(* CODESYS project Tc3_XtsInterface.library
   TcLibraryId: Beckhoff Automation GmbH|Tc3_XtsInterface|0.2.15.0
   Company: Beckhoff Automation GmbH
   Title: Tc3_XtsInterface
   Version: 0.2.15.0

Project tree, tasks and I/O mapping:
  POUs/
    Environment/
      ProcessingUnit/
        Mover/
          function block FB_XtsXlMover [ST]: FB_init, FB_exit, Init, GetParameter, SetParameter, GetObjectId, Environment, ProcessingUnit, GetActiveTrackObjectId, SetActiveTrackObjectId, GetConfiguredDetectionTrackObjectId, SetConfiguredDetectionTrackObjectId, GetStartupTrackPosition, SetStartupTrackPosition, TriggerLeave, TriggerArrive, GetSimulatedStartUpPart, SetSimulatedStartUpPart, GetSimulatedStartUpPosition, SetSimulatedStartUpPosition, GetIsVirtualFeedbackEnabled, SetIsVirtualFeedbackEnabled, GetIsDetectionOnStartupEnabled, GetIsActive, GetPositionInfo_partPosition, GetPositionInfo_trackPosition, GetPositionInfo_partObjectId, GetPositionInfo_trackObjectId, GetBtn, GetCurrentModuleCount, GetAxisId, GetAxisObjectId, GetDistanceDriven, GetDistanceDrivenInKm, GetHasDriveError, GetMoverControllerError, GetDriveStatus, GetDriveControlValue, GetMoverController, SetMoverController, GetVersion_Major, GetVersion_Minor, GetVersion_Build, GetVersion_Revision
        Part/
          Module/
            function block FB_XtsXlModule [ST]: FB_init, FB_exit, Init, GetParameter, SetParameter, GetObjectId, Environment, Part, GetIsDcLinkVoltageReady, GetVersion_Major, GetVersion_Minor, GetVersion_Build, GetVersion_Revision
          function block FB_XtsXlPart [ST]: FB_init, FB_exit, Init, GetParameter, SetParameter, GetObjectId, Environment, ModuleCount, Module, ModuleWithOid, ProcessingUnit, GetMcTrackOid, GetLength, TriggerReset, GetIsDcLinkVoltageReady, GetDriveState, GetGlobalNumber, GetVersion_Major, GetVersion_Minor, GetVersion_Build, GetVersion_Revision
        Track/
          function block FB_XtsTrack [ST]: FB_init, FB_exit, Init, GetParameter, SetParameter, GetObjectId, Environment, PartConfigCount, GetPartConfigOidAt, ProcessingUnit, GetIsClosed, GetPolarity, GetOffset, GetIsIncludedInDetection, GetDetectionPriority, GetLength, GetVersion_Major, GetVersion_Minor, GetVersion_Build, GetVersion_Revision
        function block FB_XtsProcessingUnit [ST]: FB_init, FB_exit, Init, GetParameter, SetParameter, GetObjectId, Environment, XlMoverCount, XlMover, XlMoverWithOid, XlPartCount, XlPart, XlPartWithOid, TrackCount, Track, TrackWithOid, GetActiveMoverCount, GetDriveState, GetIsDcLinkVoltageReady, GetVersion_Major, GetVersion_Minor, GetVersion_Build, GetVersion_Revision
      function block FB_XtsEnvironment [ST]: FB_init, FB_exit, Init, ProcessingUnitCount, ProcessingUnit, ProcessingUnitWithOid
  Version/
    global variables Global_Version
*)

// Version/Global_Version
{attribute 'TcGenerated'}
// This function has been automatically generated from the project information.
VAR_GLOBAL CONSTANT
	{attribute 'const_non_replaced'}
	{attribute 'linkalways'}
	stLibVersion_Tc3_XtsInterface : ST_LibVersion := (iMajor := 0, iMinor := 2, iBuild := 15, iRevision := 0, nFlags := 0, sVersion := '0.2.15.0');
	{attribute 'const_non_replaced'}
	{attribute 'linkalways'}
	sLibraryId_Tc3_XtsInterface : String := 'Beckhoff Automation GmbH|Tc3_XtsInterface|0.2.15.0';
END_VAR

// POUs/Environment/FB_XtsEnvironment

{attribute 'c++_compatible'}
{attribute 'external_name' := 'FB_XtsEnvironment_GUID_43DC2321_88A6_68C5_F281_B52FDA472D50'}
{attribute 'TcIecLibraryType'}
FUNCTION_BLOCK FB_XtsEnvironment
VAR
	 {attribute 'hide'}
	_reserved1 : ARRAY [1..12] OF UINT_8_16;
END_VAR

{attribute 'TcTypeSystem'}

(* Internal method *)
{attribute 'hide'}
METHOD FB_init : BOOL
VAR_INPUT
	(* If TRUE, the retain variables are initialized (warm start / cold start) *)
	bInitRetains : BOOL;
	(* If TRUE, the instance afterwards gets moved into the copy code (online change) *)
	bInCopyCode : BOOL;
END_VAR
END_METHOD

{attribute 'TcTypeSystem'}

(* Internal method *)
{attribute 'hide'}
METHOD FB_exit : BOOL
VAR_INPUT
	(* If TRUE, the exit method is called for exiting an instance that is copied afterwards (online change). *)
	bInCopyCode : BOOL;
END_VAR
END_METHOD

{attribute 'TcTypeSystem'}

(* Initialize the XTS environment. *)
METHOD Init
VAR_INPUT
	(* Feedback for the command. Use 0 if no feedback wanted. *)
	{attribute 'GUID' := '5F1A75BA-B0CF-46E4-B9FF-8350B6E0F16A'}
	{attribute 'Namespace' := 'Tc3_XtsInterface'}
	CommandFeedback : REFERENCE TO XtsCommandFeedback;
END_VAR
END_METHOD

{attribute 'TcTypeSystem'}

(* Returns the count of the Processing Units in the Environment. *)
METHOD ProcessingUnitCount : UINT
END_METHOD

{attribute 'TcTypeSystem'}

(* Returns the I_XtsProcessingUnit at the specified index [1, ..., size] in the Environment. *)
METHOD ProcessingUnit : I_XtsProcessingUnit1
VAR_INPUT
	(* Index of the ProcessingUnit in the Environment [1, ..., size]. *)
	Index : UINT;
	(* Feedback for the command. Use 0 if no feedback wanted. *)
	{attribute 'GUID' := '5F1A75BA-B0CF-46E4-B9FF-8350B6E0F16A'}
	{attribute 'Namespace' := 'Tc3_XtsInterface'}
	CommandFeedback : REFERENCE TO XtsCommandFeedback;
END_VAR
END_METHOD

{attribute 'TcTypeSystem'}

(* Returns the I_XtsProcessingUnit with the specified Object ID. *)
METHOD ProcessingUnitWithOid : I_XtsProcessingUnit1
VAR_INPUT
	(* Index of the ProcessingUnit in the Environment [1, ..., size]. *)
	{attribute 'GUID' := '18071995-0000-0000-0000-00000000000F'}
	ObjectId : GLOBAL.OTCID;
	(* Feedback for the command. Use 0 if no feedback wanted. *)
	{attribute 'GUID' := '5F1A75BA-B0CF-46E4-B9FF-8350B6E0F16A'}
	{attribute 'Namespace' := 'Tc3_XtsInterface'}
	CommandFeedback : REFERENCE TO XtsCommandFeedback;
END_VAR
END_METHOD

END_FUNCTION_BLOCK

// POUs/Environment/ProcessingUnit/FB_XtsProcessingUnit

{attribute 'c++_compatible'}
{attribute 'external_name' := 'FB_XtsProcessingUnit_GUID_11AFE61A_C1C5_6F5D_D8AE_C0074E97D741'}
{attribute 'TcIecLibraryType'}
FUNCTION_BLOCK FB_XtsProcessingUnit
VAR
	 {attribute 'hide'}
	_reserved1 : ARRAY [1..16] OF UINT_8_16;
END_VAR

{attribute 'TcTypeSystem'}

(* Internal method *)
{attribute 'hide'}
METHOD FB_init : BOOL
VAR_INPUT
	(* If TRUE, the retain variables are initialized (warm start / cold start) *)
	bInitRetains : BOOL;
	(* If TRUE, the instance afterwards gets moved into the copy code (online change) *)
	bInCopyCode : BOOL;
END_VAR
END_METHOD

{attribute 'TcTypeSystem'}

(* Internal method *)
{attribute 'hide'}
METHOD FB_exit : BOOL
VAR_INPUT
	(* If TRUE, the exit method is called for exiting an instance that is copied afterwards (online change). *)
	bInCopyCode : BOOL;
END_VAR
END_METHOD

{attribute 'TcTypeSystem'}

(* Initialize the XTS ProcessingUnit with a specific ObjectId. *)
METHOD Init
VAR_INPUT
	(* ObjectId of the ProcessingUnit to connect. *)
	{attribute 'GUID' := '18071995-0000-0000-0000-00000000000F'}
	ObjectId : GLOBAL.OTCID;
	(* Feedback for the command. Use 0 if no feedback wanted. *)
	{attribute 'GUID' := '5F1A75BA-B0CF-46E4-B9FF-8350B6E0F16A'}
	{attribute 'Namespace' := 'Tc3_XtsInterface'}
	CommandFeedback : REFERENCE TO XtsCommandFeedback;
END_VAR
END_METHOD

{attribute 'TcTypeSystem'}

(* Get any parameter of the Processing Unit by PID. *)
METHOD GetParameter
VAR_INPUT
	(* Parameter ID of the object parameter. *)
	{attribute 'GUID' := '18071995-0000-0000-0000-00000000001C'}
	ParameterId : GLOBAL.PTCID;
	(* Max. length of the data. *)
	nData : REFERENCE TO UDINT;
	(* Pointer to the data. *)
	{attribute 'GUID' := '18071995-0000-0000-0000-000000000018'}
	pData : REFERENCE TO GLOBAL.PVOID;
	(* Feedback for the command. Use 0 if no feedback wanted. *)
	{attribute 'GUID' := '5F1A75BA-B0CF-46E4-B9FF-8350B6E0F16A'}
	{attribute 'Namespace' := 'Tc3_XtsInterface'}
	CommandFeedback : REFERENCE TO XtsCommandFeedback;
END_VAR
END_METHOD

{attribute 'TcTypeSystem'}

(* Set any parameter of the Processing Unit by PID. *)
METHOD SetParameter
VAR_INPUT
	(* Parameter-ID of the object parameter. *)
	{attribute 'GUID' := '18071995-0000-0000-0000-00000000001C'}
	ParameterId : GLOBAL.PTCID;
	(* Max. length of the data. *)
	nData : UDINT;
	(* Pointer to the data. *)
	{attribute 'GUID' := '18071995-0000-0000-0000-000000000018'}
	pData : GLOBAL.PVOID;
	(* Feedback for the command. Use 0 if no feedback wanted. *)
	{attribute 'GUID' := '5F1A75BA-B0CF-46E4-B9FF-8350B6E0F16A'}
	{attribute 'Namespace' := 'Tc3_XtsInterface'}
	CommandFeedback : REFERENCE TO XtsCommandFeedback;
END_VAR
END_METHOD

{attribute 'TcTypeSystem'}

(* Returns the object id of the object. *)
METHOD GetObjectId : GLOBAL.OTCID
END_METHOD

{attribute 'TcTypeSystem'}

(* Get the XTS Environment. *)
METHOD Environment
VAR_INPUT
	(* Pointer to the I_XtsEnvironment. *)
	{attribute 'GUID' := '18071995-0000-0000-0000-000000000018'}
	ipEnvironment : POINTER TO GLOBAL.PVOID;
END_VAR
END_METHOD

{attribute 'TcTypeSystem'}

(* Returns the count of the Movers in the Processing Unit. *)
METHOD XlMoverCount : UINT
END_METHOD

{attribute 'TcTypeSystem'}

(* Returns the I_XtsXlMover at the specified index [1, ..., size] in the Processing Unit. *)
METHOD XlMover : I_XtsXlMover1
VAR_INPUT
	(* Index of the XL Mover in the Processing Unit [1, ..., size]. *)
	Index : UINT;
	(* Feedback for the command. Use 0 if no feedback wanted. *)
	{attribute 'GUID' := '5F1A75BA-B0CF-46E4-B9FF-8350B6E0F16A'}
	{attribute 'Namespace' := 'Tc3_XtsInterface'}
	CommandFeedback : REFERENCE TO XtsCommandFeedback;
END_VAR
END_METHOD

{attribute 'TcTypeSystem'}

(* Returns the I_XtsXlMover with the specified Object ID. *)
METHOD XlMoverWithOid : I_XtsXlMover1
VAR_INPUT
	(* Object ID of the XL Mover. *)
	{attribute 'GUID' := '18071995-0000-0000-0000-00000000000F'}
	ObjectId : GLOBAL.OTCID;
	(* Feedback for the command. Use 0 if no feedback wanted. *)
	{attribute 'GUID' := '5F1A75BA-B0CF-46E4-B9FF-8350B6E0F16A'}
	{attribute 'Namespace' := 'Tc3_XtsInterface'}
	CommandFeedback : REFERENCE TO XtsCommandFeedback;
END_VAR
END_METHOD

{attribute 'TcTypeSystem'}

(* Returns the count of the XL Parts in the Processing Unit. *)
METHOD XlPartCount : UINT
END_METHOD

{attribute 'TcTypeSystem'}

(* Returns the I_XtsXlPart at the specified index [1, ..., size] in the Processing Unit. *)
METHOD XlPart : I_XtsXlPart1
VAR_INPUT
	(* Index of the XL Part in the Processing Unit [1, ..., size]. *)
	Index : UINT;
	(* Feedback for the command. Use 0 if no feedback wanted. *)
	{attribute 'GUID' := '5F1A75BA-B0CF-46E4-B9FF-8350B6E0F16A'}
	{attribute 'Namespace' := 'Tc3_XtsInterface'}
	CommandFeedback : REFERENCE TO XtsCommandFeedback;
END_VAR
END_METHOD

{attribute 'TcTypeSystem'}

(* Returns the I_XtsXlPart with the specified Object ID. *)
METHOD XlPartWithOid : I_XtsXlPart1
VAR_INPUT
	(* Object ID of the XL Part. *)
	{attribute 'GUID' := '18071995-0000-0000-0000-00000000000F'}
	ObjectId : GLOBAL.OTCID;
	(* Feedback for the command. Use 0 if no feedback wanted. *)
	{attribute 'GUID' := '5F1A75BA-B0CF-46E4-B9FF-8350B6E0F16A'}
	{attribute 'Namespace' := 'Tc3_XtsInterface'}
	CommandFeedback : REFERENCE TO XtsCommandFeedback;
END_VAR
END_METHOD

{attribute 'TcTypeSystem'}

(* Returns the count of the Tracks in the Processing Unit. *)
METHOD TrackCount : UINT
END_METHOD

{attribute 'TcTypeSystem'}

(* Returns the I_XtsTrack at the specified index [1, ..., size] in the Processing Unit. *)
METHOD Track : I_XtsTrack1
VAR_INPUT
	(* Index of the Track in the Processing Unit [1, ..., size]. *)
	Index : UINT;
	(* Feedback for the command. Use 0 if no feedback wanted. *)
	{attribute 'GUID' := '5F1A75BA-B0CF-46E4-B9FF-8350B6E0F16A'}
	{attribute 'Namespace' := 'Tc3_XtsInterface'}
	CommandFeedback : REFERENCE TO XtsCommandFeedback;
END_VAR
END_METHOD

{attribute 'TcTypeSystem'}

(* Returns the I_XtsTrack with the specified Object ID. *)
METHOD TrackWithOid : I_XtsTrack1
VAR_INPUT
	(* Object ID of the Track. *)
	{attribute 'GUID' := '18071995-0000-0000-0000-00000000000F'}
	ObjectId : GLOBAL.OTCID;
	(* Feedback for the command. Use 0 if no feedback wanted. *)
	{attribute 'GUID' := '5F1A75BA-B0CF-46E4-B9FF-8350B6E0F16A'}
	{attribute 'Namespace' := 'Tc3_XtsInterface'}
	CommandFeedback : REFERENCE TO XtsCommandFeedback;
END_VAR
END_METHOD

{attribute 'TcTypeSystem'}

(* Returns the count of active movers. *)
METHOD GetActiveMoverCount : UDINT
VAR_INPUT
	(* Feedback for the command. Use 0 if no feedback wanted. *)
	{attribute 'GUID' := '5F1A75BA-B0CF-46E4-B9FF-8350B6E0F16A'}
	{attribute 'Namespace' := 'Tc3_XtsInterface'}
	CommandFeedback : REFERENCE TO XtsCommandFeedback;
END_VAR
END_METHOD

{attribute 'TcTypeSystem'}

(* Returns the state of the drive system. *)
METHOD GetDriveState : XTS.DriveState
VAR_INPUT
	(* Feedback for the command. Use 0 if no feedback wanted. *)
	{attribute 'GUID' := '5F1A75BA-B0CF-46E4-B9FF-8350B6E0F16A'}
	{attribute 'Namespace' := 'Tc3_XtsInterface'}
	CommandFeedback : REFERENCE TO XtsCommandFeedback;
END_VAR
END_METHOD

{attribute 'TcTypeSystem'}

(* Returns true if the DC Link voltage of all modules is ready. *)
METHOD GetIsDcLinkVoltageReady : BOOL
VAR_INPUT
	(* Feedback for the command. Use 0 if no feedback wanted. *)
	{attribute 'GUID' := '5F1A75BA-B0CF-46E4-B9FF-8350B6E0F16A'}
	{attribute 'Namespace' := 'Tc3_XtsInterface'}
	CommandFeedback : REFERENCE TO XtsCommandFeedback;
END_VAR
END_METHOD

{attribute 'TcTypeSystem'}

METHOD GetVersion_Major : UDINT
VAR_INPUT
	(* Feedback for the command. Use 0 if no feedback wanted. *)
	{attribute 'GUID' := '5F1A75BA-B0CF-46E4-B9FF-8350B6E0F16A'}
	{attribute 'Namespace' := 'Tc3_XtsInterface'}
	CommandFeedback : REFERENCE TO XtsCommandFeedback;
END_VAR
END_METHOD

{attribute 'TcTypeSystem'}

METHOD GetVersion_Minor : UDINT
VAR_INPUT
	(* Feedback for the command. Use 0 if no feedback wanted. *)
	{attribute 'GUID' := '5F1A75BA-B0CF-46E4-B9FF-8350B6E0F16A'}
	{attribute 'Namespace' := 'Tc3_XtsInterface'}
	CommandFeedback : REFERENCE TO XtsCommandFeedback;
END_VAR
END_METHOD

{attribute 'TcTypeSystem'}

METHOD GetVersion_Build : UDINT
VAR_INPUT
	(* Feedback for the command. Use 0 if no feedback wanted. *)
	{attribute 'GUID' := '5F1A75BA-B0CF-46E4-B9FF-8350B6E0F16A'}
	{attribute 'Namespace' := 'Tc3_XtsInterface'}
	CommandFeedback : REFERENCE TO XtsCommandFeedback;
END_VAR
END_METHOD

{attribute 'TcTypeSystem'}

METHOD GetVersion_Revision : UDINT
VAR_INPUT
	(* Feedback for the command. Use 0 if no feedback wanted. *)
	{attribute 'GUID' := '5F1A75BA-B0CF-46E4-B9FF-8350B6E0F16A'}
	{attribute 'Namespace' := 'Tc3_XtsInterface'}
	CommandFeedback : REFERENCE TO XtsCommandFeedback;
END_VAR
END_METHOD

END_FUNCTION_BLOCK

// POUs/Environment/ProcessingUnit/Mover/FB_XtsXlMover

{attribute 'c++_compatible'}
{attribute 'external_name' := 'FB_XtsXlMover_GUID_1E637CC7_4B33_663F_E76F_825CECCC1ED4'}
{attribute 'TcIecLibraryType'}
FUNCTION_BLOCK FB_XtsXlMover
VAR
	 {attribute 'hide'}
	_reserved1 : ARRAY [1..16] OF UINT_8_16;
END_VAR

{attribute 'TcTypeSystem'}

(* Internal method *)
{attribute 'hide'}
METHOD FB_init : BOOL
VAR_INPUT
	(* If TRUE, the retain variables are initialized (warm start / cold start) *)
	bInitRetains : BOOL;
	(* If TRUE, the instance afterwards gets moved into the copy code (online change) *)
	bInCopyCode : BOOL;
END_VAR
END_METHOD

{attribute 'TcTypeSystem'}

(* Internal method *)
{attribute 'hide'}
METHOD FB_exit : BOOL
VAR_INPUT
	(* If TRUE, the exit method is called for exiting an instance that is copied afterwards (online change). *)
	bInCopyCode : BOOL;
END_VAR
END_METHOD

{attribute 'TcTypeSystem'}

(* Initialize the XTS Mover with a specific ObjectId. *)
METHOD Init
VAR_INPUT
	(* ObjectId of the XL Mover to connect. *)
	{attribute 'GUID' := '18071995-0000-0000-0000-00000000000F'}
	ObjectId : GLOBAL.OTCID;
	(* Feedback for the command. Use 0 if no feedback wanted. *)
	{attribute 'GUID' := '5F1A75BA-B0CF-46E4-B9FF-8350B6E0F16A'}
	{attribute 'Namespace' := 'Tc3_XtsInterface'}
	CommandFeedback : REFERENCE TO XtsCommandFeedback;
END_VAR
END_METHOD

{attribute 'TcTypeSystem'}

(* Get any parameter of the Processing Unit by PID. *)
METHOD GetParameter
VAR_INPUT
	(* Parameter ID of the object parameter. *)
	{attribute 'GUID' := '18071995-0000-0000-0000-00000000001C'}
	ParameterId : GLOBAL.PTCID;
	(* Max. length of the data. *)
	nData : REFERENCE TO UDINT;
	(* Pointer to the data. *)
	{attribute 'GUID' := '18071995-0000-0000-0000-000000000018'}
	pData : REFERENCE TO GLOBAL.PVOID;
	(* Feedback for the command. Use 0 if no feedback wanted. *)
	{attribute 'GUID' := '5F1A75BA-B0CF-46E4-B9FF-8350B6E0F16A'}
	{attribute 'Namespace' := 'Tc3_XtsInterface'}
	CommandFeedback : REFERENCE TO XtsCommandFeedback;
END_VAR
END_METHOD

{attribute 'TcTypeSystem'}

(* Set any parameter of the Processing Unit by PID. *)
METHOD SetParameter
VAR_INPUT
	(* Parameter-ID of the object parameter. *)
	{attribute 'GUID' := '18071995-0000-0000-0000-00000000001C'}
	ParameterId : GLOBAL.PTCID;
	(* Max. length of the data. *)
	nData : UDINT;
	(* Pointer to the data. *)
	{attribute 'GUID' := '18071995-0000-0000-0000-000000000018'}
	pData : GLOBAL.PVOID;
	(* Feedback for the command. Use 0 if no feedback wanted. *)
	{attribute 'GUID' := '5F1A75BA-B0CF-46E4-B9FF-8350B6E0F16A'}
	{attribute 'Namespace' := 'Tc3_XtsInterface'}
	CommandFeedback : REFERENCE TO XtsCommandFeedback;
END_VAR
END_METHOD

{attribute 'TcTypeSystem'}

(* Returns the object id of the object. *)
METHOD GetObjectId : GLOBAL.OTCID
END_METHOD

{attribute 'TcTypeSystem'}

(* Get the XTS Environment. *)
METHOD Environment
VAR_INPUT
	(* Pointer to the I_XtsEnvironment. *)
	{attribute 'GUID' := '18071995-0000-0000-0000-000000000018'}
	ipEnvironment : POINTER TO GLOBAL.PVOID;
END_VAR
END_METHOD

{attribute 'TcTypeSystem'}

(* Get the parent XTS Processing Unit. *)
METHOD ProcessingUnit
VAR_INPUT
	(* Pointer to the I_XtsProcessingUnit. *)
	{attribute 'GUID' := '18071995-0000-0000-0000-000000000018'}
	ipProcessingUnit : POINTER TO GLOBAL.PVOID;
END_VAR
END_METHOD

{attribute 'TcTypeSystem'}

(* Gets/Sets the Track object Id that is currently active /should be activated for the Mover. *)
METHOD GetActiveTrackObjectId : XTS.TrackOTCID
VAR_INPUT
	(* Feedback for the command. Use 0 if no feedback wanted. *)
	{attribute 'GUID' := '5F1A75BA-B0CF-46E4-B9FF-8350B6E0F16A'}
	{attribute 'Namespace' := 'Tc3_XtsInterface'}
	CommandFeedback : REFERENCE TO XtsCommandFeedback;
END_VAR
END_METHOD

{attribute 'TcTypeSystem'}

(* Gets/Sets the Track object Id that is currently active /should be activated for the Mover. *)
METHOD SetActiveTrackObjectId
VAR_INPUT
	(* New value for ActiveTrackObjectId *)
	{attribute 'GUID' := '831FA102-5DFA-4739-AD9A-80CFCA3F6F7A'}
	{attribute 'Namespace' := 'XTS'}
	ActiveTrackObjectId : XTS.TrackOTCID;
	(* Feedback for the command. Use 0 if no feedback wanted. *)
	{attribute 'GUID' := '5F1A75BA-B0CF-46E4-B9FF-8350B6E0F16A'}
	{attribute 'Namespace' := 'Tc3_XtsInterface'}
	CommandFeedback : REFERENCE TO XtsCommandFeedback;
END_VAR
END_METHOD

{attribute 'TcTypeSystem'}

(* Gets/Sets the Track object Id on which the detection is executed when the arrive is triggered. *)
METHOD GetConfiguredDetectionTrackObjectId : XTS.TrackOTCID
VAR_INPUT
	(* Feedback for the command. Use 0 if no feedback wanted. *)
	{attribute 'GUID' := '5F1A75BA-B0CF-46E4-B9FF-8350B6E0F16A'}
	{attribute 'Namespace' := 'Tc3_XtsInterface'}
	CommandFeedback : REFERENCE TO XtsCommandFeedback;
END_VAR
END_METHOD

{attribute 'TcTypeSystem'}

(* Gets/Sets the Track object Id on which the detection is executed when the arrive is triggered. *)
METHOD SetConfiguredDetectionTrackObjectId
VAR_INPUT
	(* New value for ConfiguredDetectionTrackObjectId *)
	{attribute 'GUID' := '831FA102-5DFA-4739-AD9A-80CFCA3F6F7A'}
	{attribute 'Namespace' := 'XTS'}
	ConfiguredDetectionTrackObjectId : XTS.TrackOTCID;
	(* Feedback for the command. Use 0 if no feedback wanted. *)
	{attribute 'GUID' := '5F1A75BA-B0CF-46E4-B9FF-8350B6E0F16A'}
	{attribute 'Namespace' := 'Tc3_XtsInterface'}
	CommandFeedback : REFERENCE TO XtsCommandFeedback;
END_VAR
END_METHOD

{attribute 'TcTypeSystem'}

(* Without multiturn detection you have to define a position on the track with a tolerance of +-24mm. *)
METHOD GetStartupTrackPosition : REAL
VAR_INPUT
	(* Feedback for the command. Use 0 if no feedback wanted. *)
	{attribute 'GUID' := '5F1A75BA-B0CF-46E4-B9FF-8350B6E0F16A'}
	{attribute 'Namespace' := 'Tc3_XtsInterface'}
	CommandFeedback : REFERENCE TO XtsCommandFeedback;
END_VAR
END_METHOD

{attribute 'TcTypeSystem'}

(* Without multiturn detection you have to define a position on the track with a tolerance of +-24mm. *)
METHOD SetStartupTrackPosition
VAR_INPUT
	(* New value for StartupTrackPosition *)
	StartupTrackPosition : REAL;
	(* Feedback for the command. Use 0 if no feedback wanted. *)
	{attribute 'GUID' := '5F1A75BA-B0CF-46E4-B9FF-8350B6E0F16A'}
	{attribute 'Namespace' := 'Tc3_XtsInterface'}
	CommandFeedback : REFERENCE TO XtsCommandFeedback;
END_VAR
END_METHOD

{attribute 'TcTypeSystem'}

(* If downloaded then the active is set to passive. The mover cannot be used anymore - it is ready to leave the system without any error. *)
METHOD TriggerLeave
VAR_INPUT
	(* Feedback for the command. Use 0 if no feedback wanted. *)
	{attribute 'GUID' := '5F1A75BA-B0CF-46E4-B9FF-8350B6E0F16A'}
	{attribute 'Namespace' := 'Tc3_XtsInterface'}
	CommandFeedback : REFERENCE TO XtsCommandFeedback;
END_VAR
END_METHOD

{attribute 'TcTypeSystem'}

(* If downloaded then a detection for one mover on the configured track is executed if successful the mover is activated. *)
METHOD TriggerArrive
VAR_INPUT
	(* Feedback for the command. Use 0 if no feedback wanted. *)
	{attribute 'GUID' := '5F1A75BA-B0CF-46E4-B9FF-8350B6E0F16A'}
	{attribute 'Namespace' := 'Tc3_XtsInterface'}
	CommandFeedback : REFERENCE TO XtsCommandFeedback;
END_VAR
END_METHOD

{attribute 'TcTypeSystem'}

(* Gets/sets the part on which the mover is detected during simulation. *)
METHOD GetSimulatedStartUpPart : XTS.XlPartOTCID
VAR_INPUT
	(* Feedback for the command. Use 0 if no feedback wanted. *)
	{attribute 'GUID' := '5F1A75BA-B0CF-46E4-B9FF-8350B6E0F16A'}
	{attribute 'Namespace' := 'Tc3_XtsInterface'}
	CommandFeedback : REFERENCE TO XtsCommandFeedback;
END_VAR
END_METHOD

{attribute 'TcTypeSystem'}

(* Gets/sets the part on which the mover is detected during simulation. *)
METHOD SetSimulatedStartUpPart
VAR_INPUT
	(* New value for SimulatedStartUpPart *)
	{attribute 'GUID' := '77AA1C52-88B2-44B0-8ADB-666DDD3510A0'}
	{attribute 'Namespace' := 'XTS'}
	SimulatedStartUpPart : XTS.XlPartOTCID;
	(* Feedback for the command. Use 0 if no feedback wanted. *)
	{attribute 'GUID' := '5F1A75BA-B0CF-46E4-B9FF-8350B6E0F16A'}
	{attribute 'Namespace' := 'Tc3_XtsInterface'}
	CommandFeedback : REFERENCE TO XtsCommandFeedback;
END_VAR
END_METHOD

{attribute 'TcTypeSystem'}

(* Gets/sets the part on which the mover is detected during simulation. *)
METHOD GetSimulatedStartUpPosition : LREAL
VAR_INPUT
	(* Feedback for the command. Use 0 if no feedback wanted. *)
	{attribute 'GUID' := '5F1A75BA-B0CF-46E4-B9FF-8350B6E0F16A'}
	{attribute 'Namespace' := 'Tc3_XtsInterface'}
	CommandFeedback : REFERENCE TO XtsCommandFeedback;
END_VAR
END_METHOD

{attribute 'TcTypeSystem'}

(* Gets/sets the part on which the mover is detected during simulation. *)
METHOD SetSimulatedStartUpPosition
VAR_INPUT
	(* New value for SimulatedStartUpPosition *)
	SimulatedStartUpPosition : LREAL;
	(* Feedback for the command. Use 0 if no feedback wanted. *)
	{attribute 'GUID' := '5F1A75BA-B0CF-46E4-B9FF-8350B6E0F16A'}
	{attribute 'Namespace' := 'Tc3_XtsInterface'}
	CommandFeedback : REFERENCE TO XtsCommandFeedback;
END_VAR
END_METHOD

{attribute 'TcTypeSystem'}

(* If enabled the actual position follows the setPosition ignoring missing hardware. *)
METHOD GetIsVirtualFeedbackEnabled : BOOL
VAR_INPUT
	(* Feedback for the command. Use 0 if no feedback wanted. *)
	{attribute 'GUID' := '5F1A75BA-B0CF-46E4-B9FF-8350B6E0F16A'}
	{attribute 'Namespace' := 'Tc3_XtsInterface'}
	CommandFeedback : REFERENCE TO XtsCommandFeedback;
END_VAR
END_METHOD

{attribute 'TcTypeSystem'}

(* If enabled the actual position follows the setPosition ignoring missing hardware. *)
METHOD SetIsVirtualFeedbackEnabled
VAR_INPUT
	(* New value for IsVirtualFeedbackEnabled *)
	IsVirtualFeedbackEnabled : BOOL;
	(* Feedback for the command. Use 0 if no feedback wanted. *)
	{attribute 'GUID' := '5F1A75BA-B0CF-46E4-B9FF-8350B6E0F16A'}
	{attribute 'Namespace' := 'Tc3_XtsInterface'}
	CommandFeedback : REFERENCE TO XtsCommandFeedback;
END_VAR
END_METHOD

{attribute 'TcTypeSystem'}

(* If true the mover is detected on the StartupTrack with the configured StartupTrackPosition. *)
METHOD GetIsDetectionOnStartupEnabled : BOOL
VAR_INPUT
	(* Feedback for the command. Use 0 if no feedback wanted. *)
	{attribute 'GUID' := '5F1A75BA-B0CF-46E4-B9FF-8350B6E0F16A'}
	{attribute 'Namespace' := 'Tc3_XtsInterface'}
	CommandFeedback : REFERENCE TO XtsCommandFeedback;
END_VAR
END_METHOD

{attribute 'TcTypeSystem'}

(* Gets value which indicates if the mover is actively used or is currently passive. An active mover may be deactivated if one plans to remove it from the system. *)
METHOD GetIsActive : BOOL
VAR_INPUT
	(* Feedback for the command. Use 0 if no feedback wanted. *)
	{attribute 'GUID' := '5F1A75BA-B0CF-46E4-B9FF-8350B6E0F16A'}
	{attribute 'Namespace' := 'Tc3_XtsInterface'}
	CommandFeedback : REFERENCE TO XtsCommandFeedback;
END_VAR
END_METHOD

{attribute 'TcTypeSystem'}

METHOD GetPositionInfo_partPosition : LREAL
VAR_INPUT
	(* Feedback for the command. Use 0 if no feedback wanted. *)
	{attribute 'GUID' := '5F1A75BA-B0CF-46E4-B9FF-8350B6E0F16A'}
	{attribute 'Namespace' := 'Tc3_XtsInterface'}
	CommandFeedback : REFERENCE TO XtsCommandFeedback;
END_VAR
END_METHOD

{attribute 'TcTypeSystem'}

METHOD GetPositionInfo_trackPosition : LREAL
VAR_INPUT
	(* Feedback for the command. Use 0 if no feedback wanted. *)
	{attribute 'GUID' := '5F1A75BA-B0CF-46E4-B9FF-8350B6E0F16A'}
	{attribute 'Namespace' := 'Tc3_XtsInterface'}
	CommandFeedback : REFERENCE TO XtsCommandFeedback;
END_VAR
END_METHOD

{attribute 'TcTypeSystem'}

METHOD GetPositionInfo_partObjectId : GLOBAL.OTCID
VAR_INPUT
	(* Feedback for the command. Use 0 if no feedback wanted. *)
	{attribute 'GUID' := '5F1A75BA-B0CF-46E4-B9FF-8350B6E0F16A'}
	{attribute 'Namespace' := 'Tc3_XtsInterface'}
	CommandFeedback : REFERENCE TO XtsCommandFeedback;
END_VAR
END_METHOD

{attribute 'TcTypeSystem'}

METHOD GetPositionInfo_trackObjectId : GLOBAL.OTCID
VAR_INPUT
	(* Feedback for the command. Use 0 if no feedback wanted. *)
	{attribute 'GUID' := '5F1A75BA-B0CF-46E4-B9FF-8350B6E0F16A'}
	{attribute 'Namespace' := 'Tc3_XtsInterface'}
	CommandFeedback : REFERENCE TO XtsCommandFeedback;
END_VAR
END_METHOD

{attribute 'TcTypeSystem'}

(* Returns the BTN of the mover. *)
METHOD GetBtn : XTS.Btn
VAR_INPUT
	(* Feedback for the command. Use 0 if no feedback wanted. *)
	{attribute 'GUID' := '5F1A75BA-B0CF-46E4-B9FF-8350B6E0F16A'}
	{attribute 'Namespace' := 'Tc3_XtsInterface'}
	CommandFeedback : REFERENCE TO XtsCommandFeedback;
END_VAR
END_METHOD

{attribute 'TcTypeSystem'}

(* Returns the number of modules. *)
METHOD GetCurrentModuleCount : UDINT
VAR_INPUT
	(* Feedback for the command. Use 0 if no feedback wanted. *)
	{attribute 'GUID' := '5F1A75BA-B0CF-46E4-B9FF-8350B6E0F16A'}
	{attribute 'Namespace' := 'Tc3_XtsInterface'}
	CommandFeedback : REFERENCE TO XtsCommandFeedback;
END_VAR
END_METHOD

{attribute 'TcTypeSystem'}

(* Gets the ID of the associated axis. *)
METHOD GetAxisId : UDINT
VAR_INPUT
	(* Feedback for the command. Use 0 if no feedback wanted. *)
	{attribute 'GUID' := '5F1A75BA-B0CF-46E4-B9FF-8350B6E0F16A'}
	{attribute 'Namespace' := 'Tc3_XtsInterface'}
	CommandFeedback : REFERENCE TO XtsCommandFeedback;
END_VAR
END_METHOD

{attribute 'TcTypeSystem'}

(* Gets the object ID of the associated axis. *)
METHOD GetAxisObjectId : GLOBAL.OTCID
VAR_INPUT
	(* Feedback for the command. Use 0 if no feedback wanted. *)
	{attribute 'GUID' := '5F1A75BA-B0CF-46E4-B9FF-8350B6E0F16A'}
	{attribute 'Namespace' := 'Tc3_XtsInterface'}
	CommandFeedback : REFERENCE TO XtsCommandFeedback;
END_VAR
END_METHOD

{attribute 'TcTypeSystem'}

(* Returns the value of the absolute distance driven by the mover in mm. *)
METHOD GetDistanceDriven : LREAL
VAR_INPUT
	(* Feedback for the command. Use 0 if no feedback wanted. *)
	{attribute 'GUID' := '5F1A75BA-B0CF-46E4-B9FF-8350B6E0F16A'}
	{attribute 'Namespace' := 'Tc3_XtsInterface'}
	CommandFeedback : REFERENCE TO XtsCommandFeedback;
END_VAR
END_METHOD

{attribute 'TcTypeSystem'}

(* Returns the value of the absolute distance driven by the mover in km. *)
METHOD GetDistanceDrivenInKm : LREAL
VAR_INPUT
	(* Feedback for the command. Use 0 if no feedback wanted. *)
	{attribute 'GUID' := '5F1A75BA-B0CF-46E4-B9FF-8350B6E0F16A'}
	{attribute 'Namespace' := 'Tc3_XtsInterface'}
	CommandFeedback : REFERENCE TO XtsCommandFeedback;
END_VAR
END_METHOD

{attribute 'TcTypeSystem'}

(* Returns true if the motor module which is used by a mover signals an error. *)
METHOD GetHasDriveError : GLOBAL.BOOL32
VAR_INPUT
	(* Feedback for the command. Use 0 if no feedback wanted. *)
	{attribute 'GUID' := '5F1A75BA-B0CF-46E4-B9FF-8350B6E0F16A'}
	{attribute 'Namespace' := 'Tc3_XtsInterface'}
	CommandFeedback : REFERENCE TO XtsCommandFeedback;
END_VAR
END_METHOD

{attribute 'TcTypeSystem'}

(* Returns the error code of the linked XTS Mover Controller. *)
METHOD GetMoverControllerError : UINT
VAR_INPUT
	(* Feedback for the command. Use 0 if no feedback wanted. *)
	{attribute 'GUID' := '5F1A75BA-B0CF-46E4-B9FF-8350B6E0F16A'}
	{attribute 'Namespace' := 'Tc3_XtsInterface'}
	CommandFeedback : REFERENCE TO XtsCommandFeedback;
END_VAR
END_METHOD

{attribute 'TcTypeSystem'}

(* Returns the drive status of the mover. *)
METHOD GetDriveStatus : XTS.DriveState
VAR_INPUT
	(* Feedback for the command. Use 0 if no feedback wanted. *)
	{attribute 'GUID' := '5F1A75BA-B0CF-46E4-B9FF-8350B6E0F16A'}
	{attribute 'Namespace' := 'Tc3_XtsInterface'}
	CommandFeedback : REFERENCE TO XtsCommandFeedback;
END_VAR
END_METHOD

{attribute 'TcTypeSystem'}

(* Returns the drive control value of the mover. *)
METHOD GetDriveControlValue : UINT
VAR_INPUT
	(* Feedback for the command. Use 0 if no feedback wanted. *)
	{attribute 'GUID' := '5F1A75BA-B0CF-46E4-B9FF-8350B6E0F16A'}
	{attribute 'Namespace' := 'Tc3_XtsInterface'}
	CommandFeedback : REFERENCE TO XtsCommandFeedback;
END_VAR
END_METHOD

{attribute 'TcTypeSystem'}

(* Get/set the the mover controller. *)
METHOD GetMoverController : XTS.XtsMoverControllerOTCID
VAR_INPUT
	(* Feedback for the command. Use 0 if no feedback wanted. *)
	{attribute 'GUID' := '5F1A75BA-B0CF-46E4-B9FF-8350B6E0F16A'}
	{attribute 'Namespace' := 'Tc3_XtsInterface'}
	CommandFeedback : REFERENCE TO XtsCommandFeedback;
END_VAR
END_METHOD

{attribute 'TcTypeSystem'}

(* Get/set the the mover controller. *)
METHOD SetMoverController
VAR_INPUT
	(* New value for MoverController *)
	{attribute 'GUID' := '01E5C78E-D451-4377-9F02-F3812CC92C14'}
	{attribute 'Namespace' := 'XTS'}
	MoverController : XTS.XtsMoverControllerOTCID;
	(* Feedback for the command. Use 0 if no feedback wanted. *)
	{attribute 'GUID' := '5F1A75BA-B0CF-46E4-B9FF-8350B6E0F16A'}
	{attribute 'Namespace' := 'Tc3_XtsInterface'}
	CommandFeedback : REFERENCE TO XtsCommandFeedback;
END_VAR
END_METHOD

{attribute 'TcTypeSystem'}

METHOD GetVersion_Major : UDINT
VAR_INPUT
	(* Feedback for the command. Use 0 if no feedback wanted. *)
	{attribute 'GUID' := '5F1A75BA-B0CF-46E4-B9FF-8350B6E0F16A'}
	{attribute 'Namespace' := 'Tc3_XtsInterface'}
	CommandFeedback : REFERENCE TO XtsCommandFeedback;
END_VAR
END_METHOD

{attribute 'TcTypeSystem'}

METHOD GetVersion_Minor : UDINT
VAR_INPUT
	(* Feedback for the command. Use 0 if no feedback wanted. *)
	{attribute 'GUID' := '5F1A75BA-B0CF-46E4-B9FF-8350B6E0F16A'}
	{attribute 'Namespace' := 'Tc3_XtsInterface'}
	CommandFeedback : REFERENCE TO XtsCommandFeedback;
END_VAR
END_METHOD

{attribute 'TcTypeSystem'}

METHOD GetVersion_Build : UDINT
VAR_INPUT
	(* Feedback for the command. Use 0 if no feedback wanted. *)
	{attribute 'GUID' := '5F1A75BA-B0CF-46E4-B9FF-8350B6E0F16A'}
	{attribute 'Namespace' := 'Tc3_XtsInterface'}
	CommandFeedback : REFERENCE TO XtsCommandFeedback;
END_VAR
END_METHOD

{attribute 'TcTypeSystem'}

METHOD GetVersion_Revision : UDINT
VAR_INPUT
	(* Feedback for the command. Use 0 if no feedback wanted. *)
	{attribute 'GUID' := '5F1A75BA-B0CF-46E4-B9FF-8350B6E0F16A'}
	{attribute 'Namespace' := 'Tc3_XtsInterface'}
	CommandFeedback : REFERENCE TO XtsCommandFeedback;
END_VAR
END_METHOD

END_FUNCTION_BLOCK

// POUs/Environment/ProcessingUnit/Part/FB_XtsXlPart

{attribute 'c++_compatible'}
{attribute 'external_name' := 'FB_XtsXlPart_GUID_4DA3CFA6_2547_65DA_DBE8_E66BFF8BF8A4'}
{attribute 'TcIecLibraryType'}
FUNCTION_BLOCK FB_XtsXlPart
VAR
	 {attribute 'hide'}
	_reserved1 : ARRAY [1..16] OF UINT_8_16;
END_VAR

{attribute 'TcTypeSystem'}

(* Internal method *)
{attribute 'hide'}
METHOD FB_init : BOOL
VAR_INPUT
	(* If TRUE, the retain variables are initialized (warm start / cold start) *)
	bInitRetains : BOOL;
	(* If TRUE, the instance afterwards gets moved into the copy code (online change) *)
	bInCopyCode : BOOL;
END_VAR
END_METHOD

{attribute 'TcTypeSystem'}

(* Internal method *)
{attribute 'hide'}
METHOD FB_exit : BOOL
VAR_INPUT
	(* If TRUE, the exit method is called for exiting an instance that is copied afterwards (online change). *)
	bInCopyCode : BOOL;
END_VAR
END_METHOD

{attribute 'TcTypeSystem'}

(* Initialize the XTS XL Part with a specific ObjectId. *)
METHOD Init
VAR_INPUT
	(* ObjectId of the XL Part to connect. *)
	{attribute 'GUID' := '18071995-0000-0000-0000-00000000000F'}
	ObjectId : GLOBAL.OTCID;
	(* Feedback for the command. Use 0 if no feedback wanted. *)
	{attribute 'GUID' := '5F1A75BA-B0CF-46E4-B9FF-8350B6E0F16A'}
	{attribute 'Namespace' := 'Tc3_XtsInterface'}
	CommandFeedback : REFERENCE TO XtsCommandFeedback;
END_VAR
END_METHOD

{attribute 'TcTypeSystem'}

(* Get any parameter of the Processing Unit by PID. *)
METHOD GetParameter
VAR_INPUT
	(* Parameter ID of the object parameter. *)
	{attribute 'GUID' := '18071995-0000-0000-0000-00000000001C'}
	ParameterId : GLOBAL.PTCID;
	(* Max. length of the data. *)
	nData : REFERENCE TO UDINT;
	(* Pointer to the data. *)
	{attribute 'GUID' := '18071995-0000-0000-0000-000000000018'}
	pData : REFERENCE TO GLOBAL.PVOID;
	(* Feedback for the command. Use 0 if no feedback wanted. *)
	{attribute 'GUID' := '5F1A75BA-B0CF-46E4-B9FF-8350B6E0F16A'}
	{attribute 'Namespace' := 'Tc3_XtsInterface'}
	CommandFeedback : REFERENCE TO XtsCommandFeedback;
END_VAR
END_METHOD

{attribute 'TcTypeSystem'}

(* Set any parameter of the Processing Unit by PID. *)
METHOD SetParameter
VAR_INPUT
	(* Parameter-ID of the object parameter. *)
	{attribute 'GUID' := '18071995-0000-0000-0000-00000000001C'}
	ParameterId : GLOBAL.PTCID;
	(* Max. length of the data. *)
	nData : UDINT;
	(* Pointer to the data. *)
	{attribute 'GUID' := '18071995-0000-0000-0000-000000000018'}
	pData : GLOBAL.PVOID;
	(* Feedback for the command. Use 0 if no feedback wanted. *)
	{attribute 'GUID' := '5F1A75BA-B0CF-46E4-B9FF-8350B6E0F16A'}
	{attribute 'Namespace' := 'Tc3_XtsInterface'}
	CommandFeedback : REFERENCE TO XtsCommandFeedback;
END_VAR
END_METHOD

{attribute 'TcTypeSystem'}

(* Returns the object id of the object. *)
METHOD GetObjectId : GLOBAL.OTCID
END_METHOD

{attribute 'TcTypeSystem'}

(* Get the XTS Environment. *)
METHOD Environment
VAR_INPUT
	(* Pointer to the I_XtsEnvironment. *)
	{attribute 'GUID' := '18071995-0000-0000-0000-000000000018'}
	ipEnvironment : POINTER TO GLOBAL.PVOID;
END_VAR
END_METHOD

{attribute 'TcTypeSystem'}

(* Returns the count of the XL Modules in the XL Part. *)
METHOD ModuleCount : UINT
END_METHOD

{attribute 'TcTypeSystem'}

(* Returns the I_XtsXlModule at the specified index [1, ..., size] in the XL Part. *)
METHOD Module : I_XtsXlModule1
VAR_INPUT
	(* Index of the XL Module in the XL Part [1, ..., size]. *)
	Index : UINT;
	(* Feedback for the command. Use 0 if no feedback wanted. *)
	{attribute 'GUID' := '5F1A75BA-B0CF-46E4-B9FF-8350B6E0F16A'}
	{attribute 'Namespace' := 'Tc3_XtsInterface'}
	CommandFeedback : REFERENCE TO XtsCommandFeedback;
END_VAR
END_METHOD

{attribute 'TcTypeSystem'}

(* Returns the I_XtsXlModule with the specified Object ID. *)
METHOD ModuleWithOid : I_XtsXlModule1
VAR_INPUT
	(* Object ID of the XL Module. *)
	{attribute 'GUID' := '18071995-0000-0000-0000-00000000000F'}
	ObjectId : GLOBAL.OTCID;
	(* Feedback for the command. Use 0 if no feedback wanted. *)
	{attribute 'GUID' := '5F1A75BA-B0CF-46E4-B9FF-8350B6E0F16A'}
	{attribute 'Namespace' := 'Tc3_XtsInterface'}
	CommandFeedback : REFERENCE TO XtsCommandFeedback;
END_VAR
END_METHOD

{attribute 'TcTypeSystem'}

(* Get the parent XTS Processing Unit. *)
METHOD ProcessingUnit
VAR_INPUT
	(* Pointer to the I_XtsProcessingUnit. *)
	{attribute 'GUID' := '18071995-0000-0000-0000-000000000018'}
	ipProcessingUnit : POINTER TO GLOBAL.PVOID;
END_VAR
END_METHOD

{attribute 'TcTypeSystem'}

(* Set the corresponding McTrack. *)
METHOD GetMcTrackOid : MC.PlanarTrackOTCID
VAR_INPUT
	(* Feedback for the command. Use 0 if no feedback wanted. *)
	{attribute 'GUID' := '5F1A75BA-B0CF-46E4-B9FF-8350B6E0F16A'}
	{attribute 'Namespace' := 'Tc3_XtsInterface'}
	CommandFeedback : REFERENCE TO XtsCommandFeedback;
END_VAR
END_METHOD

{attribute 'TcTypeSystem'}

(* Set the length of the XL Part. *)
METHOD GetLength : LREAL
VAR_INPUT
	(* Feedback for the command. Use 0 if no feedback wanted. *)
	{attribute 'GUID' := '5F1A75BA-B0CF-46E4-B9FF-8350B6E0F16A'}
	{attribute 'Namespace' := 'Tc3_XtsInterface'}
	CommandFeedback : REFERENCE TO XtsCommandFeedback;
END_VAR
END_METHOD

{attribute 'TcTypeSystem'}

(* If downloaded then all faulty modules will be resetted. *)
METHOD TriggerReset
VAR_INPUT
	(* Feedback for the command. Use 0 if no feedback wanted. *)
	{attribute 'GUID' := '5F1A75BA-B0CF-46E4-B9FF-8350B6E0F16A'}
	{attribute 'Namespace' := 'Tc3_XtsInterface'}
	CommandFeedback : REFERENCE TO XtsCommandFeedback;
END_VAR
END_METHOD

{attribute 'TcTypeSystem'}

(* Returns true if the DC Link voltage of all modules is ready (requires PartBasedHandling). *)
METHOD GetIsDcLinkVoltageReady : BOOL
VAR_INPUT
	(* Feedback for the command. Use 0 if no feedback wanted. *)
	{attribute 'GUID' := '5F1A75BA-B0CF-46E4-B9FF-8350B6E0F16A'}
	{attribute 'Namespace' := 'Tc3_XtsInterface'}
	CommandFeedback : REFERENCE TO XtsCommandFeedback;
END_VAR
END_METHOD

{attribute 'TcTypeSystem'}

(* Returns the state of the drive system. *)
METHOD GetDriveState : XTS.DriveState
VAR_INPUT
	(* Feedback for the command. Use 0 if no feedback wanted. *)
	{attribute 'GUID' := '5F1A75BA-B0CF-46E4-B9FF-8350B6E0F16A'}
	{attribute 'Namespace' := 'Tc3_XtsInterface'}
	CommandFeedback : REFERENCE TO XtsCommandFeedback;
END_VAR
END_METHOD

{attribute 'TcTypeSystem'}

(* The global number is used to distinguish all parts which are manged by one XPU. *)
METHOD GetGlobalNumber : UDINT
VAR_INPUT
	(* Feedback for the command. Use 0 if no feedback wanted. *)
	{attribute 'GUID' := '5F1A75BA-B0CF-46E4-B9FF-8350B6E0F16A'}
	{attribute 'Namespace' := 'Tc3_XtsInterface'}
	CommandFeedback : REFERENCE TO XtsCommandFeedback;
END_VAR
END_METHOD

{attribute 'TcTypeSystem'}

METHOD GetVersion_Major : UDINT
VAR_INPUT
	(* Feedback for the command. Use 0 if no feedback wanted. *)
	{attribute 'GUID' := '5F1A75BA-B0CF-46E4-B9FF-8350B6E0F16A'}
	{attribute 'Namespace' := 'Tc3_XtsInterface'}
	CommandFeedback : REFERENCE TO XtsCommandFeedback;
END_VAR
END_METHOD

{attribute 'TcTypeSystem'}

METHOD GetVersion_Minor : UDINT
VAR_INPUT
	(* Feedback for the command. Use 0 if no feedback wanted. *)
	{attribute 'GUID' := '5F1A75BA-B0CF-46E4-B9FF-8350B6E0F16A'}
	{attribute 'Namespace' := 'Tc3_XtsInterface'}
	CommandFeedback : REFERENCE TO XtsCommandFeedback;
END_VAR
END_METHOD

{attribute 'TcTypeSystem'}

METHOD GetVersion_Build : UDINT
VAR_INPUT
	(* Feedback for the command. Use 0 if no feedback wanted. *)
	{attribute 'GUID' := '5F1A75BA-B0CF-46E4-B9FF-8350B6E0F16A'}
	{attribute 'Namespace' := 'Tc3_XtsInterface'}
	CommandFeedback : REFERENCE TO XtsCommandFeedback;
END_VAR
END_METHOD

{attribute 'TcTypeSystem'}

METHOD GetVersion_Revision : UDINT
VAR_INPUT
	(* Feedback for the command. Use 0 if no feedback wanted. *)
	{attribute 'GUID' := '5F1A75BA-B0CF-46E4-B9FF-8350B6E0F16A'}
	{attribute 'Namespace' := 'Tc3_XtsInterface'}
	CommandFeedback : REFERENCE TO XtsCommandFeedback;
END_VAR
END_METHOD

END_FUNCTION_BLOCK

// POUs/Environment/ProcessingUnit/Track/FB_XtsTrack

{attribute 'c++_compatible'}
{attribute 'external_name' := 'FB_XtsTrack_GUID_4A6FB3C2_4387_6806_F909_338CC0F04911'}
{attribute 'TcIecLibraryType'}
FUNCTION_BLOCK FB_XtsTrack
VAR
	 {attribute 'hide'}
	_reserved1 : ARRAY [1..16] OF UINT_8_16;
END_VAR

{attribute 'TcTypeSystem'}

(* Internal method *)
{attribute 'hide'}
METHOD FB_init : BOOL
VAR_INPUT
	(* If TRUE, the retain variables are initialized (warm start / cold start) *)
	bInitRetains : BOOL;
	(* If TRUE, the instance afterwards gets moved into the copy code (online change) *)
	bInCopyCode : BOOL;
END_VAR
END_METHOD

{attribute 'TcTypeSystem'}

(* Internal method *)
{attribute 'hide'}
METHOD FB_exit : BOOL
VAR_INPUT
	(* If TRUE, the exit method is called for exiting an instance that is copied afterwards (online change). *)
	bInCopyCode : BOOL;
END_VAR
END_METHOD

{attribute 'TcTypeSystem'}

(* Initialize the XTS Track with a specific ObjectId. *)
METHOD Init
VAR_INPUT
	(* ObjectId of the Track to connect. *)
	{attribute 'GUID' := '18071995-0000-0000-0000-00000000000F'}
	ObjectId : GLOBAL.OTCID;
	(* Feedback for the command. Use 0 if no feedback wanted. *)
	{attribute 'GUID' := '5F1A75BA-B0CF-46E4-B9FF-8350B6E0F16A'}
	{attribute 'Namespace' := 'Tc3_XtsInterface'}
	CommandFeedback : REFERENCE TO XtsCommandFeedback;
END_VAR
END_METHOD

{attribute 'TcTypeSystem'}

(* Get any parameter of the Processing Unit by PID. *)
METHOD GetParameter
VAR_INPUT
	(* Parameter ID of the object parameter. *)
	{attribute 'GUID' := '18071995-0000-0000-0000-00000000001C'}
	ParameterId : GLOBAL.PTCID;
	(* Max. length of the data. *)
	nData : REFERENCE TO UDINT;
	(* Pointer to the data. *)
	{attribute 'GUID' := '18071995-0000-0000-0000-000000000018'}
	pData : REFERENCE TO GLOBAL.PVOID;
	(* Feedback for the command. Use 0 if no feedback wanted. *)
	{attribute 'GUID' := '5F1A75BA-B0CF-46E4-B9FF-8350B6E0F16A'}
	{attribute 'Namespace' := 'Tc3_XtsInterface'}
	CommandFeedback : REFERENCE TO XtsCommandFeedback;
END_VAR
END_METHOD

{attribute 'TcTypeSystem'}

(* Set any parameter of the Processing Unit by PID. *)
METHOD SetParameter
VAR_INPUT
	(* Parameter-ID of the object parameter. *)
	{attribute 'GUID' := '18071995-0000-0000-0000-00000000001C'}
	ParameterId : GLOBAL.PTCID;
	(* Max. length of the data. *)
	nData : UDINT;
	(* Pointer to the data. *)
	{attribute 'GUID' := '18071995-0000-0000-0000-000000000018'}
	pData : GLOBAL.PVOID;
	(* Feedback for the command. Use 0 if no feedback wanted. *)
	{attribute 'GUID' := '5F1A75BA-B0CF-46E4-B9FF-8350B6E0F16A'}
	{attribute 'Namespace' := 'Tc3_XtsInterface'}
	CommandFeedback : REFERENCE TO XtsCommandFeedback;
END_VAR
END_METHOD

{attribute 'TcTypeSystem'}

(* Returns the object id of the object. *)
METHOD GetObjectId : GLOBAL.OTCID
END_METHOD

{attribute 'TcTypeSystem'}

(* Get the XTS Environment. *)
METHOD Environment
VAR_INPUT
	(* Pointer to the I_XtsEnvironment. *)
	{attribute 'GUID' := '18071995-0000-0000-0000-000000000018'}
	ipEnvironment : POINTER TO GLOBAL.PVOID;
END_VAR
END_METHOD

{attribute 'TcTypeSystem'}

(* Returns the count of the PartConfigs in the Track. *)
METHOD PartConfigCount : UINT
END_METHOD

{attribute 'TcTypeSystem'}

(* Returns the OTCID of the Part at the specified index [1, ..., size] in the Track. *)
METHOD GetPartConfigOidAt : GLOBAL.OTCID
VAR_INPUT
	(* Index of the PartConfig in the Track [1, ..., size]. *)
	Index : UINT;
	(* Feedback for the command. Use 0 if no feedback wanted. *)
	{attribute 'GUID' := '5F1A75BA-B0CF-46E4-B9FF-8350B6E0F16A'}
	{attribute 'Namespace' := 'Tc3_XtsInterface'}
	CommandFeedback : REFERENCE TO XtsCommandFeedback;
END_VAR
END_METHOD

{attribute 'TcTypeSystem'}

(* Get the parent XTS Processing Unit. *)
METHOD ProcessingUnit
VAR_INPUT
	(* Pointer to the I_XtsProcessingUnit. *)
	{attribute 'GUID' := '18071995-0000-0000-0000-000000000018'}
	ipProcessingUnit : POINTER TO GLOBAL.PVOID;
END_VAR
END_METHOD

{attribute 'TcTypeSystem'}

(* Configure if the Track is closed. *)
METHOD GetIsClosed : BOOL
VAR_INPUT
	(* Feedback for the command. Use 0 if no feedback wanted. *)
	{attribute 'GUID' := '5F1A75BA-B0CF-46E4-B9FF-8350B6E0F16A'}
	{attribute 'Namespace' := 'Tc3_XtsInterface'}
	CommandFeedback : REFERENCE TO XtsCommandFeedback;
END_VAR
END_METHOD

{attribute 'TcTypeSystem'}

(* Configure the direction of the part. Only positive is supported at the moment. *)
METHOD GetPolarity : XTS.Polarity
VAR_INPUT
	(* Feedback for the command. Use 0 if no feedback wanted. *)
	{attribute 'GUID' := '5F1A75BA-B0CF-46E4-B9FF-8350B6E0F16A'}
	{attribute 'Namespace' := 'Tc3_XtsInterface'}
	CommandFeedback : REFERENCE TO XtsCommandFeedback;
END_VAR
END_METHOD

{attribute 'TcTypeSystem'}

(* Configure the offset for the Track. *)
METHOD GetOffset : LREAL
VAR_INPUT
	(* Feedback for the command. Use 0 if no feedback wanted. *)
	{attribute 'GUID' := '5F1A75BA-B0CF-46E4-B9FF-8350B6E0F16A'}
	{attribute 'Namespace' := 'Tc3_XtsInterface'}
	CommandFeedback : REFERENCE TO XtsCommandFeedback;
END_VAR
END_METHOD

{attribute 'TcTypeSystem'}

(* Configure if this Track is included in the Mover detection. *)
METHOD GetIsIncludedInDetection : BOOL
VAR_INPUT
	(* Feedback for the command. Use 0 if no feedback wanted. *)
	{attribute 'GUID' := '5F1A75BA-B0CF-46E4-B9FF-8350B6E0F16A'}
	{attribute 'Namespace' := 'Tc3_XtsInterface'}
	CommandFeedback : REFERENCE TO XtsCommandFeedback;
END_VAR
END_METHOD

{attribute 'TcTypeSystem'}

(* Set the priority for the Mover detection on this Track. *)
METHOD GetDetectionPriority : UDINT
VAR_INPUT
	(* Feedback for the command. Use 0 if no feedback wanted. *)
	{attribute 'GUID' := '5F1A75BA-B0CF-46E4-B9FF-8350B6E0F16A'}
	{attribute 'Namespace' := 'Tc3_XtsInterface'}
	CommandFeedback : REFERENCE TO XtsCommandFeedback;
END_VAR
END_METHOD

{attribute 'TcTypeSystem'}

(* Returns the length of the Track. *)
METHOD GetLength : LREAL
VAR_INPUT
	(* Feedback for the command. Use 0 if no feedback wanted. *)
	{attribute 'GUID' := '5F1A75BA-B0CF-46E4-B9FF-8350B6E0F16A'}
	{attribute 'Namespace' := 'Tc3_XtsInterface'}
	CommandFeedback : REFERENCE TO XtsCommandFeedback;
END_VAR
END_METHOD

{attribute 'TcTypeSystem'}

METHOD GetVersion_Major : UDINT
VAR_INPUT
	(* Feedback for the command. Use 0 if no feedback wanted. *)
	{attribute 'GUID' := '5F1A75BA-B0CF-46E4-B9FF-8350B6E0F16A'}
	{attribute 'Namespace' := 'Tc3_XtsInterface'}
	CommandFeedback : REFERENCE TO XtsCommandFeedback;
END_VAR
END_METHOD

{attribute 'TcTypeSystem'}

METHOD GetVersion_Minor : UDINT
VAR_INPUT
	(* Feedback for the command. Use 0 if no feedback wanted. *)
	{attribute 'GUID' := '5F1A75BA-B0CF-46E4-B9FF-8350B6E0F16A'}
	{attribute 'Namespace' := 'Tc3_XtsInterface'}
	CommandFeedback : REFERENCE TO XtsCommandFeedback;
END_VAR
END_METHOD

{attribute 'TcTypeSystem'}

METHOD GetVersion_Build : UDINT
VAR_INPUT
	(* Feedback for the command. Use 0 if no feedback wanted. *)
	{attribute 'GUID' := '5F1A75BA-B0CF-46E4-B9FF-8350B6E0F16A'}
	{attribute 'Namespace' := 'Tc3_XtsInterface'}
	CommandFeedback : REFERENCE TO XtsCommandFeedback;
END_VAR
END_METHOD

{attribute 'TcTypeSystem'}

METHOD GetVersion_Revision : UDINT
VAR_INPUT
	(* Feedback for the command. Use 0 if no feedback wanted. *)
	{attribute 'GUID' := '5F1A75BA-B0CF-46E4-B9FF-8350B6E0F16A'}
	{attribute 'Namespace' := 'Tc3_XtsInterface'}
	CommandFeedback : REFERENCE TO XtsCommandFeedback;
END_VAR
END_METHOD

END_FUNCTION_BLOCK

// POUs/Environment/ProcessingUnit/Part/Module/FB_XtsXlModule

{attribute 'c++_compatible'}
{attribute 'external_name' := 'FB_XtsXlModule_GUID_BA974C8F_3779_6ABF_DBA7_E88B8C065BC5'}
{attribute 'TcIecLibraryType'}
FUNCTION_BLOCK FB_XtsXlModule
VAR
	 {attribute 'hide'}
	_reserved1 : ARRAY [1..16] OF UINT_8_16;
END_VAR

{attribute 'TcTypeSystem'}

(* Internal method *)
{attribute 'hide'}
METHOD FB_init : BOOL
VAR_INPUT
	(* If TRUE, the retain variables are initialized (warm start / cold start) *)
	bInitRetains : BOOL;
	(* If TRUE, the instance afterwards gets moved into the copy code (online change) *)
	bInCopyCode : BOOL;
END_VAR
END_METHOD

{attribute 'TcTypeSystem'}

(* Internal method *)
{attribute 'hide'}
METHOD FB_exit : BOOL
VAR_INPUT
	(* If TRUE, the exit method is called for exiting an instance that is copied afterwards (online change). *)
	bInCopyCode : BOOL;
END_VAR
END_METHOD

{attribute 'TcTypeSystem'}

(* Initialize the XTS XL Module with a specific ObjectId. *)
METHOD Init
VAR_INPUT
	(* ObjectId of the XL Module to connect. *)
	{attribute 'GUID' := '18071995-0000-0000-0000-00000000000F'}
	ObjectId : GLOBAL.OTCID;
	(* Feedback for the command. Use 0 if no feedback wanted. *)
	{attribute 'GUID' := '5F1A75BA-B0CF-46E4-B9FF-8350B6E0F16A'}
	{attribute 'Namespace' := 'Tc3_XtsInterface'}
	CommandFeedback : REFERENCE TO XtsCommandFeedback;
END_VAR
END_METHOD

{attribute 'TcTypeSystem'}

(* Get any parameter of the Processing Unit by PID. *)
METHOD GetParameter
VAR_INPUT
	(* Parameter ID of the object parameter. *)
	{attribute 'GUID' := '18071995-0000-0000-0000-00000000001C'}
	ParameterId : GLOBAL.PTCID;
	(* Max. length of the data. *)
	nData : REFERENCE TO UDINT;
	(* Pointer to the data. *)
	{attribute 'GUID' := '18071995-0000-0000-0000-000000000018'}
	pData : REFERENCE TO GLOBAL.PVOID;
	(* Feedback for the command. Use 0 if no feedback wanted. *)
	{attribute 'GUID' := '5F1A75BA-B0CF-46E4-B9FF-8350B6E0F16A'}
	{attribute 'Namespace' := 'Tc3_XtsInterface'}
	CommandFeedback : REFERENCE TO XtsCommandFeedback;
END_VAR
END_METHOD

{attribute 'TcTypeSystem'}

(* Set any parameter of the Processing Unit by PID. *)
METHOD SetParameter
VAR_INPUT
	(* Parameter-ID of the object parameter. *)
	{attribute 'GUID' := '18071995-0000-0000-0000-00000000001C'}
	ParameterId : GLOBAL.PTCID;
	(* Max. length of the data. *)
	nData : UDINT;
	(* Pointer to the data. *)
	{attribute 'GUID' := '18071995-0000-0000-0000-000000000018'}
	pData : GLOBAL.PVOID;
	(* Feedback for the command. Use 0 if no feedback wanted. *)
	{attribute 'GUID' := '5F1A75BA-B0CF-46E4-B9FF-8350B6E0F16A'}
	{attribute 'Namespace' := 'Tc3_XtsInterface'}
	CommandFeedback : REFERENCE TO XtsCommandFeedback;
END_VAR
END_METHOD

{attribute 'TcTypeSystem'}

(* Returns the object id of the object. *)
METHOD GetObjectId : GLOBAL.OTCID
END_METHOD

{attribute 'TcTypeSystem'}

(* Get the XTS Environment. *)
METHOD Environment
VAR_INPUT
	(* Pointer to the I_XtsEnvironment. *)
	{attribute 'GUID' := '18071995-0000-0000-0000-000000000018'}
	ipEnvironment : POINTER TO GLOBAL.PVOID;
END_VAR
END_METHOD

{attribute 'TcTypeSystem'}

(* Get the parent XTS XL Part. *)
METHOD Part
VAR_INPUT
	(* Pointer to the I_XtsXlPart. *)
	{attribute 'GUID' := '18071995-0000-0000-0000-000000000018'}
	ipPart : POINTER TO GLOBAL.PVOID;
END_VAR
END_METHOD

{attribute 'TcTypeSystem'}

(* Returns true if 'DC Link Voltage' is higher or equal 'MinDcLinkVoltage'. *)
METHOD GetIsDcLinkVoltageReady : BOOL
VAR_INPUT
	(* Feedback for the command. Use 0 if no feedback wanted. *)
	{attribute 'GUID' := '5F1A75BA-B0CF-46E4-B9FF-8350B6E0F16A'}
	{attribute 'Namespace' := 'Tc3_XtsInterface'}
	CommandFeedback : REFERENCE TO XtsCommandFeedback;
END_VAR
END_METHOD

{attribute 'TcTypeSystem'}

METHOD GetVersion_Major : UDINT
VAR_INPUT
	(* Feedback for the command. Use 0 if no feedback wanted. *)
	{attribute 'GUID' := '5F1A75BA-B0CF-46E4-B9FF-8350B6E0F16A'}
	{attribute 'Namespace' := 'Tc3_XtsInterface'}
	CommandFeedback : REFERENCE TO XtsCommandFeedback;
END_VAR
END_METHOD

{attribute 'TcTypeSystem'}

METHOD GetVersion_Minor : UDINT
VAR_INPUT
	(* Feedback for the command. Use 0 if no feedback wanted. *)
	{attribute 'GUID' := '5F1A75BA-B0CF-46E4-B9FF-8350B6E0F16A'}
	{attribute 'Namespace' := 'Tc3_XtsInterface'}
	CommandFeedback : REFERENCE TO XtsCommandFeedback;
END_VAR
END_METHOD

{attribute 'TcTypeSystem'}

METHOD GetVersion_Build : UDINT
VAR_INPUT
	(* Feedback for the command. Use 0 if no feedback wanted. *)
	{attribute 'GUID' := '5F1A75BA-B0CF-46E4-B9FF-8350B6E0F16A'}
	{attribute 'Namespace' := 'Tc3_XtsInterface'}
	CommandFeedback : REFERENCE TO XtsCommandFeedback;
END_VAR
END_METHOD

{attribute 'TcTypeSystem'}

METHOD GetVersion_Revision : UDINT
VAR_INPUT
	(* Feedback for the command. Use 0 if no feedback wanted. *)
	{attribute 'GUID' := '5F1A75BA-B0CF-46E4-B9FF-8350B6E0F16A'}
	{attribute 'Namespace' := 'Tc3_XtsInterface'}
	CommandFeedback : REFERENCE TO XtsCommandFeedback;
END_VAR
END_METHOD

END_FUNCTION_BLOCK
